// Mitsubishi GX Works2 project: Memorytest   PLC: Q02U

PROGRAM MAIN
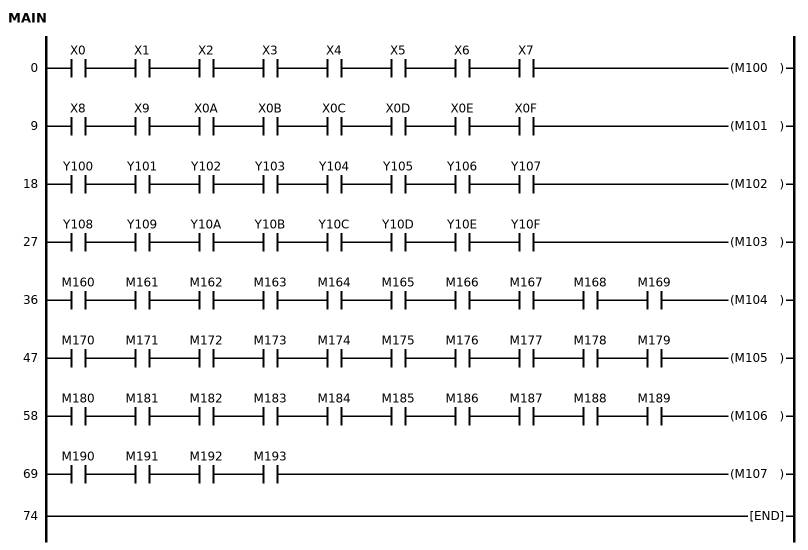
0     LD      X0
      AND     X1
      AND     X2
      AND     X3
      AND     X4
      AND     X5
      AND     X6
      AND     X7
      OUT     M100
9     LD      X8
      AND     X9
      AND     X0A
      AND     X0B
      AND     X0C
      AND     X0D
      AND     X0E
      AND     X0F
      OUT     M101
18    LD      Y100
      AND     Y101
      AND     Y102
      AND     Y103
      AND     Y104
      AND     Y105
      AND     Y106
      AND     Y107
      OUT     M102
27    LD      Y108
      AND     Y109
      AND     Y10A
      AND     Y10B
      AND     Y10C
      AND     Y10D
      AND     Y10E
      AND     Y10F
      OUT     M103
36    LD      M160
      AND     M161
      AND     M162
      AND     M163
      AND     M164
      AND     M165
      AND     M166
      AND     M167
      AND     M168
      AND     M169
      OUT     M104
47    LD      M170
      AND     M171
      AND     M172
      AND     M173
      AND     M174
      AND     M175
      AND     M176
      AND     M177
      AND     M178
      AND     M179
      OUT     M105
58    LD      M180
      AND     M181
      AND     M182
      AND     M183
      AND     M184
      AND     M185
      AND     M186
      AND     M187
      AND     M188
      AND     M189
      OUT     M106
69    LD      M190
      AND     M191
      AND     M192
      AND     M193
      OUT     M107
74    END
END_PROGRAM
